// TIA Portal V20 export
DATA_BLOCK "CC_Vibrating_Unit_1"   // DB33, Motion_DB
// stored: AutoNumber false, InstanceOfName TO_SpeedAxis, OfSystemLibElement TO_SpeedAxis, OfSystemLibVersion 7.0
TO_SpeedAxis   // technology object, version 7.0
// stored: Connection Interface Actor, InputAddress 3568, OutputAddress 3560
   // // inherited from TO_Axis
   // // inherited from TO_Object
   // VAR
   //    Velocity { ExternalWritable := 'False'} : LReal;
   //    Acceleration { ExternalWritable := 'False'} : LReal;
   //    ActualSpeed { ExternalWritable := 'False'} : LReal;
   //    VelocitySetpoint { ExternalWritable := 'False'} : LReal;
   //    Actor { S7_SetPoint := 'True'} : TO_Struct_Actor;
   //    TorqueLimiting { S7_SetPoint := 'True'} : TO_Struct_TorqueLimiting;
   //    LoadGear { S7_SetPoint := 'True'} : TO_Struct_LoadGear;
   //    DynamicLimits { S7_SetPoint := 'True'} : TO_Struct_DynamicLimits;
   //    DynamicDefaults { S7_SetPoint := 'True'} : TO_Struct_DynamicDefaults;
   //    Override { S7_SetPoint := 'True'} : TO_Struct_Override;
   //    Units { ExternalWritable := 'False'; S7_SetPoint := 'True'} : TO_Struct_Units;
   //    StatusDrive { ExternalWritable := 'False'; S7_SetPoint := 'True'} : TO_Struct_StatusDrive;
   //    StatusTorqueData { ExternalWritable := 'False'; S7_SetPoint := 'True'} : TO_Struct_StatusTorqueData;
   //    StatusMotionIn { ExternalWritable := 'False'; S7_SetPoint := 'True'} : TO_Struct_StatusMotionIn;
   //    StatusWord { ExternalWritable := 'False'} : DWord;
   //    StatusWord2 { ExternalWritable := 'False'} : DWord;
   //    ErrorWord { ExternalWritable := 'False'} : DWord;
   //    ErrorDetail { ExternalWritable := 'False'; S7_SetPoint := 'True'} : TO_Struct_ErrorDetail;
   //    WarningWord { ExternalWritable := 'False'} : DWord;
   //    ControlPanel { S7_SetPoint := 'True'} : TO_Struct_ControlPanel;
   //    InternalToTrace { S7_SetPoint := 'True'} : Array[1..4] of TO_Struct_Internal;
   //    VirtualAxis { ExternalWritable := 'False'; S7_SetPoint := 'True'} : TO_Struct_VirtualAxis;
   //    Simulation { S7_SetPoint := 'True'} : TO_Struct_AxisSimulation;
   // END_VAR
BEGIN
   Actor.DataAdaption := 1;
   Actor.Interface.AddressIn.RID := 16#2080708;
   Actor.Interface.AddressIn.AREA := 16#81;
   Actor.Interface.AddressIn.OFFSET := 3568;
   Actor.Interface.AddressOut.RID := 16#2080709;
   Actor.Interface.AddressOut.AREA := 16#82;
   Actor.Interface.AddressOut.OFFSET := 3560;
   Actor.DriveParameter.ReferenceSpeed := 2840.0;
   Actor.DriveParameter.ReferenceTorque := 18.8296;
   DynamicLimits.MaxAcceleration := 1000.0;
   DynamicLimits.MaxDeceleration := 1000.0;
   DynamicLimits.MaxJerk := 20000.0;
   DynamicDefaults.Velocity := 3000.0;
   DynamicDefaults.Acceleration := 16.6666666666667;
   DynamicDefaults.Deceleration := 16.6666666666667;
   DynamicDefaults.Jerk := 333.333333333333;
   DynamicDefaults.EmergencyDeceleration := 1000.0;
   _Actor.Interface.Telegram := 1;
   _Actor.DataAdaptionOffline := True;
END_DATA_BLOCK
